PROGRAM prgTestStatistics
VAR
	statistics:FB_BasicStatsFuns;
	aStats: ARRAY [1..7] OF LREAL := [15, 12, 11, 7, -5, 33, 45];
	avg: LREAL;
	maxi: LREAL;
	mini: LREAL;
	range: LREAL;
	variance: LREAL;
	std:LREAL;
END_VAR

avg:= statistics.M_Avg(aStats);

maxi:=statistics.M_Max(aStats);

mini:= statistics.M_Min(aStats);

range:= statistics.M_Range(aStats);

variance:=statistics.M_Variance(aStats);

std:= statistics.M_Std(aStats);

END_PROGRAM

(* stored: Version 1.1.0.1, ProductVersion 3.1.4024.12
   POU prgTestStatistics: Id {406d69a2-6a89-4950-9b4e-88b0bafeda65}, SpecialFunc None *)
